// TIA Portal V19 export
TYPE "LEXCHANGETRAY_typeConstraintRollerEm_recieve_interface"
// stored: Access Published
   STRUCT
      roller { S7_SetPoint := 'True'} : "LEXCHANGETRAY_typeConstraintRollerEm_toRollerRecieve";
      constraintWorkstation { S7_SetPoint := 'True'} : "LEXCHANGETRAY_typeConstraintRollerEm_toConstraintWorkstationRecieve";
      handlingXyz { S7_SetPoint := 'True'} : "LEXCHANGETRAY_typeConstraintRollerEm_toHandlingXyzRecieve";
   END_STRUCT;
END_TYPE
